(* PLC project Unnamed, Unknown Unnamed 1 *)
(* stored: creationDateTime 2026-01-05T10:12:26, modificationDateTime 2026-01-05T10:12:26 *)

PROGRAM main
  VAR_INPUT
    X0 : BOOL;
    X1 : BOOL;
    X2 : BOOL;
  END_VAR
  VAR_OUTPUT
    Y0 : BOOL;
    Y1 : BOOL;
    Y2 : BOOL;
  END_VAR

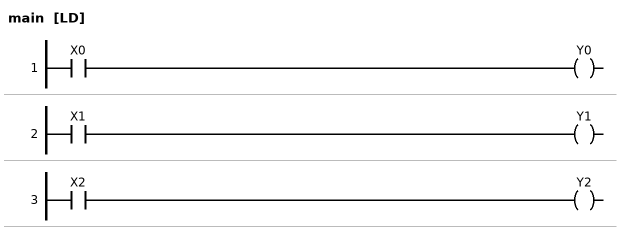
(* LD diagram, written out as Structured Text *)
Y0 := X0;
Y1 := X1;
Y2 := X2;
END_PROGRAM

CONFIGURATION Config0
  RESOURCE Res0 ON PLC
    TASK task0(INTERVAL := T#20ms, PRIORITY := 1);
    PROGRAM instance0 WITH task0 : main;
  END_RESOURCE
END_CONFIGURATION
